{attribute 'linkalways'} 
{attribute 'no_explicit_call' := 'This FB is a CLASS and must be accessed using methods or properties'}
{attribute 'enable_dynamic_creation'}
FUNCTION_BLOCK Node_F_VN_PointToLineDistance_TcVnPoint2_REAL EXTENDS VisionNode
VAR
    aPoint : _TcVnPoint2_REAL;
    aLinePoint1 : _TcVnPoint2_REAL;
    aLinePoint2 : _TcVnPoint2_REAL;
    fDistance : _LREAL(0.0);
    hrPrev : _HRESULT(S_OK);
	hresult : _HRESULT(S_OK);
END_VAR

METHOD PUBLIC  Clone : I_Node
VAR
	pNode : POINTER TO Node_F_VN_PointToLineDistance_TcVnPoint2_REAL;
END_VAR
pNode := __NEW(Node_F_VN_PointToLineDistance_TcVnPoint2_REAL);
Clone := pNode^;
END_METHOD

METHOD FB_init : BOOL
VAR_INPUT
	bInitRetains : BOOL; // if TRUE, the retain variables are initialized (warm start / cold start)
	bInCopyCode : BOOL;  // if TRUE, the instance afterwards gets moved into the copy code (online change)
END_VAR
AddInput('aPoint', aPoint);
AddInput('aLinePoint1', aLinePoint1);
AddInput('aLinePoint2', aLinePoint2);
AddInput('hrPrev', hrPrev);
AddOutput('fDistance', fDistance);
AddOutput('hresult',hresult);
END_METHOD

METHOD PROTECTED OnExecute
hresult.Value := F_VN_PointToLineDistance_TcVnPoint2_REAL(
	aPoint := aPoint.Value,
    aLinePoint1 := aLinePoint1.Value,
    aLinePoint2 := aLinePoint2.Value,
    fDistance := fDistance.Value,
	hrPrev:= hrPrev.Value);
END_METHOD

METHOD PUBLIC PreExecutionCheck
VAR_INPUT
	Check : I_PreExecutionChecks;
END_VAR
END_METHOD

END_FUNCTION_BLOCK

(* stored: Version 1.1.0.1, ProductVersion 3.1.4024.15
   POU Node_F_VN_PointToLineDistance_TcVnPoint2_REAL: Id {fa4ea7cd-e175-0217-2243-e3b50fab8339}, SpecialFunc None
   Folder Constructor: Id {b0349096-264e-05cd-1112-9e0fd7d16574}
   Method Clone: Id {49949164-8078-033a-3f16-8886da5a473e}
   Method FB_init: Id {a68e7695-0af2-0be8-0483-d4532435aa2a}
   Method OnExecute: Id {d24c93cc-6021-0125-0a26-be445b205ed4}
   Method PreExecutionCheck: Id {d5540911-ca47-02f7-2476-714fa58381ed} *)
